// TwinCAT 3 PLC project PLCsim
// ProgramVersion: 3.1.4026.20
// CompilerDefines: VISU_USEPROPERTYINFO
// libraries:
//   Tc2_Standard, * (Beckhoff Automation GmbH)
//   Tc2_System, * (Beckhoff Automation GmbH)
//   VisuSymbols, 4.5.0.0 (System)
// project tree:
//   / GlobalTextList.TcGTLO, PlcTask.TcTTO (not stored), Visualization Manager.TcVMO (not stored)
//   GVLs/ GVL.TcGVL
//   POUs/ MAIN.TcPOU
//   VISUs/ Visualization.TcVIS
// (motion and I/O tree: see PLC project plcstudent)
// real-time tasks:
//   TASK PlcTask: cycle T#10ms, priority 20, ADS port 350
//   TASK PlcTask1: cycle T#10ms, priority 21, ADS port 351
// variable links:
//   PLCsim/PLCsim Instance <-> PLCstudent/PLCstudent Instance
//     PlcTask Inputs/GVL.isStatusText <-> PlcTask Outputs/GVL.qsStatusText
//     PlcTask Inputs/GVL.iwPumpSpeed <-> PlcTask Outputs/GVL.qwPumpSpeed
//     PlcTask Outputs/GVL.qwActualLevel <-> PlcTask Inputs/GVL.iwActualLevel

// ---- GVLs/GVL.TcGVL
{attribute 'qualified_only'}
VAR_GLOBAL
	iwPumpSpeed   		AT%I* :  WORD; 	// Speed of the flow into the tank 0 - 100%
										// 40% slowly drain 50% stand still 60% filling
										

	isStatusText 		AT%I* : STRING := 'Test text'; // Text on the info display
	
	qwActualLevel 		AT%Q* : WORD;  	// Level in the tank	
	
END_VAR

// ---- POUs/MAIN.TcPOU
PROGRAM MAIN
VAR
	mwTankLevel: WORD;
	mxPumpOn: BOOL;
	mrTankLevel: REAL;
	mxOpenDrainingValve: BOOL;
END_VAR



mxPumpOn := GVL.iwPumpSpeed > 0;


IF mxOpenDrainingValve THEN
	mrTankLevel := mrTankLevel - 0.5;
END_IF

mrTankLevel :=  mrTankLevel + GVL.iwPumpSpeed/100.0;




IF (mrTankLevel < 0) THEN
	mrTankLevel := 0;
END_IF

IF (mrTankLevel > 300) THEN
	mrTankLevel := 300;
END_IF


mwTankLevel := REAL_TO_WORD( mrTankLevel);

gvl.qwActualLevel := REAL_TO_WORD(mwTankLevel / 3);

END_PROGRAM

// ---- GlobalTextList.TcGTLO
TEXTLIST GlobalTextList
  592 = '0%'
  809 = '100%'
  569 = '50%'
  694 = 'M'
  588 = 'Status Info'
  25 = 'Status: %S'
  282 = 'Status: %s'
  431 = 'Water outlet'
END_TEXTLIST

// ---- VISUs/Visualization.TcVIS
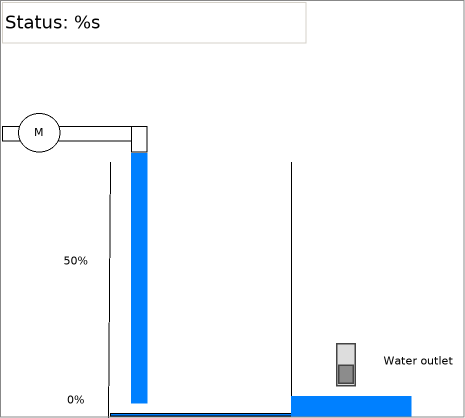
VISUALIZATION Visualization  // 465x418
    RoundedRectangle (110,413 182x3)
        p2773130477: - MAIN.mwTankLevel
    Textfield (2,2 304x41), "Status: %s", text variable: GVL.isStatusText
    Line (291,162) (291,415)
    Line (110,162) (108,418)
    Rectangle (2,126 145x15)
    Rectangle (131,126 16x26)
    Ellipse (18,113 42x39), "M"
    Rectangle (131,153 16x250), invisible if: Not MAIN.mxPumpOn
    Rectangle (291,396 120x20), invisible if: Not Main.mxOpenDrainingValve
    DipSwitch (318,343 56x43), variable: MAIN.mxOpenDrainingValve, behaviour: TOGGLE, style: Switch-DipSwitch-Gray
    Label (48,243 56x36), "50%"
    Label (48,382 56x36), "0%"
    Label (372,343 93x36), "Water outlet"
END_VISUALIZATION
